Fanuc KAREL source: compact_preamble.KL

PROGRAM KT00090
%NOLOCKGROUP
VAR
H1 : ARRAY[2] OF SHORT
I2:INTEGER
OUT:REAL
BEGIN
H1[1]=2
I2=3
OUT=((H1[1] * I2))
END KT00090
